(* PLC project MotionTest1, Higen MCL 1 *)
(* stored: creationDateTime 2012-01-06T15:20:13, modificationDateTime 2013-04-12T19:32:27 *)

FUNCTION_BLOCK wxgetval
  VAR
    getpy : python_gear;
    latch : SR;
  END_VAR
  VAR_INPUT
    name : STRING;
  END_VAR
  VAR_OUTPUT
    val : BOOL;
  END_VAR
  VAR  (* added by the conversion: wires and edge detectors of the diagram *)
    _EQ41_ENO : BOOL;
    _EQ41_OUT : BOOL;
    _EQ3_ENO : BOOL;
    _EQ3_OUT : BOOL;
  END_VAR

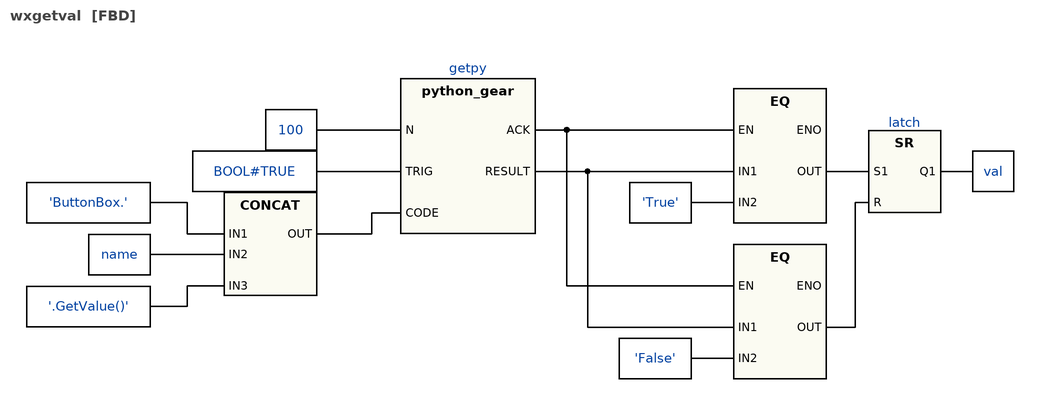
(* FBD diagram, written out as Structured Text *)
getpy(N := 100, TRIG := BOOL#TRUE, CODE := CONCAT('ButtonBox.', name, '.GetValue()'));
_EQ41_OUT := EQ(EN := getpy.ACK, IN1 := getpy.RESULT, IN2 := 'True', ENO => _EQ41_ENO);
_EQ3_OUT := EQ(EN := getpy.ACK, IN1 := getpy.RESULT, IN2 := 'False', ENO => _EQ3_ENO);
latch(S1 := _EQ41_OUT, R := _EQ3_OUT);
val := latch.Q1;
END_FUNCTION_BLOCK

(* -- *)
PROGRAM main
  VAR
    Done : BOOL;
    Slave : AXIS_REF;
    Master : AXIS_REF;
    switch : MC_Power;
    readpos : MC_ReadActualPosition;
    sPn : LREAL;
    mPn : LREAL;
    sVn : LREAL;
    mVn : LREAL;
    setpos : MC_SetPosition;
    readspeed : MC_ReadParameter;
    sim : MC_Sim;
    bt1 : wxgetval;
    Block1 : wxgetval;
    Block2 : wxgetval;
    Block3 : wxgetval;
    Block6 : wxgetval;
    Block4 : wxgetval;
    Block7 : wxgetval;
    MC_Sim0 : MC_Sim;
    MC_Power0 : MC_Power;
    MC_ReadActualPosition0 : MC_ReadActualPosition;
    MC_SetPosition0 : MC_SetPosition;
    MC_ReadParameter0 : MC_ReadParameter;
    MC_MoveAbsolute0 : MC_MoveAbsolute;
    MC_CAM_REF_FROM_CSV0 : MC_CAM_REF_FROM_CSV;
    MC_CamTableSelect0 : MC_CamTableSelect;
    MC_CamIn0 : MC_CamIn;
    MC_CamOut0 : MC_CamOut;
  END_VAR

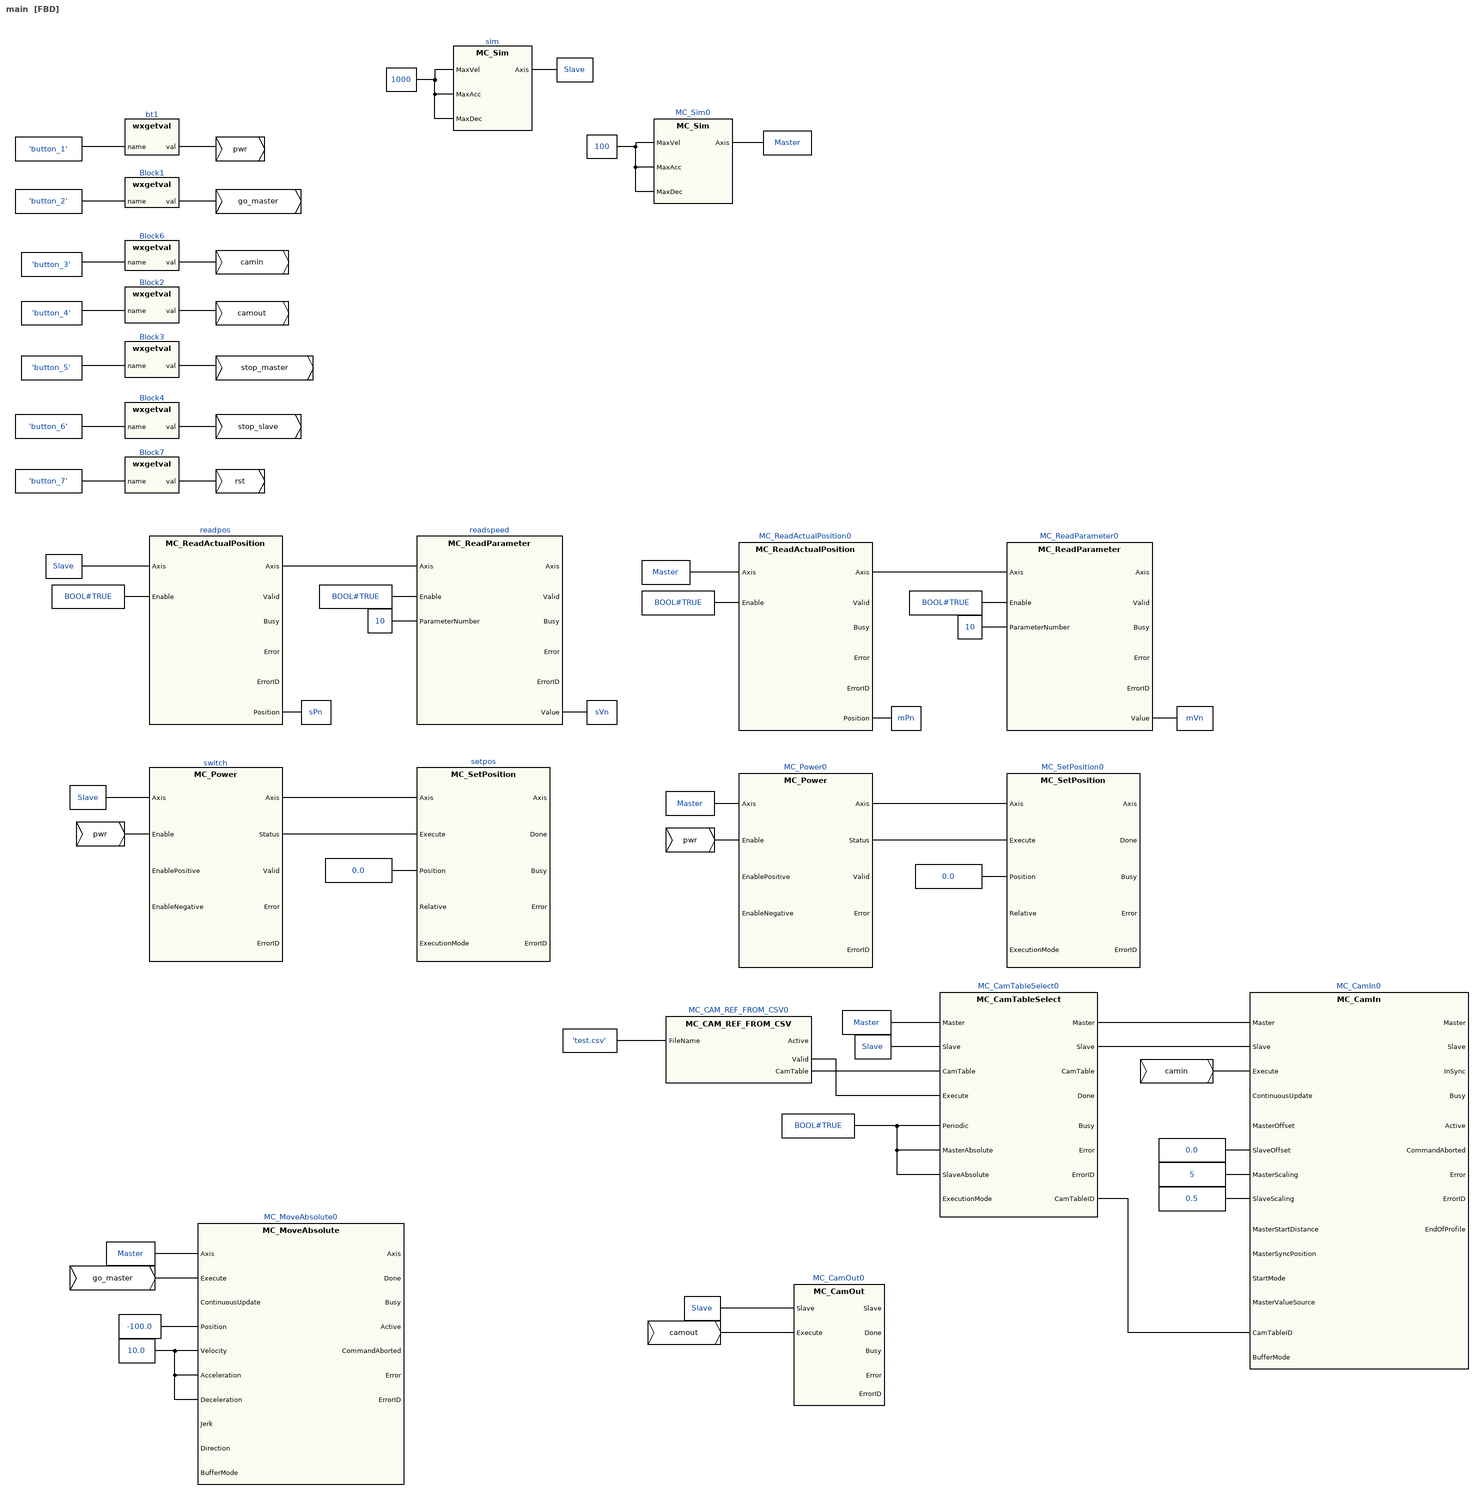
(* FBD diagram, written out as Structured Text *)
sim(MaxVel := 1000, MaxAcc := 1000, MaxDec := 1000);
Slave := sim.Axis;
MC_Sim0(MaxVel := 100, MaxAcc := 100, MaxDec := 100);
Master := MC_Sim0.Axis;
readpos(Axis := Slave, Enable := BOOL#TRUE);
sPn := readpos.Position;
readspeed(Axis := readpos.Axis, Enable := BOOL#TRUE, ParameterNumber := 10);
sVn := readspeed.Value;
MC_ReadActualPosition0(Axis := Master, Enable := BOOL#TRUE);
mPn := MC_ReadActualPosition0.Position;
MC_ReadParameter0(Axis := MC_ReadActualPosition0.Axis, Enable := BOOL#TRUE, ParameterNumber := 10);
mVn := MC_ReadParameter0.Value;
bt1(name := 'button_1');
Block1(name := 'button_2');
Block6(name := 'button_3');
Block2(name := 'button_4');
Block3(name := 'button_5');
Block4(name := 'button_6');
Block7(name := 'button_7');
switch(Axis := Slave, Enable := bt1.val);
setpos(Axis := switch.Axis, Execute := switch.Status, Position := 0.0);
MC_Power0(Axis := Master, Enable := bt1.val);
MC_SetPosition0(Axis := MC_Power0.Axis, Execute := MC_Power0.Status, Position := 0.0);
MC_CAM_REF_FROM_CSV0(FileName := 'test.csv');
MC_CamTableSelect0(Master := Master, Slave := Slave, CamTable := MC_CAM_REF_FROM_CSV0.CamTable, Execute := MC_CAM_REF_FROM_CSV0.Valid, Periodic := BOOL#TRUE, MasterAbsolute := BOOL#TRUE, SlaveAbsolute := BOOL#TRUE);
MC_CamIn0(Master := MC_CamTableSelect0.Master, Slave := MC_CamTableSelect0.Slave, Execute := Block6.val, SlaveOffset := 0.0, MasterScaling := 5, SlaveScaling := 0.5, CamTableID := MC_CamTableSelect0.CamTableID);
MC_MoveAbsolute0(Axis := Master, Execute := Block1.val, Position := -100.0, Velocity := 10.0, Acceleration := 10.0, Deceleration := 10.0);
MC_CamOut0(Slave := Slave, Execute := Block2.val);
END_PROGRAM

CONFIGURATION conf
  RESOURCE res ON PLC
    TASK milisecond(INTERVAL := T#10ms, PRIORITY := 0);
    PROGRAM maininstance WITH milisecond : main;
  END_RESOURCE
END_CONFIGURATION
